///////////
// Structure for CtrlPcs Jema .  
//////////
TYPE PCS_Jema :
STRUCT
// PCS Controller  Measures
	AX_PowerCol					: ARRAY[1..3] OF PowerCol;

	MesData						: PCS ; 
	
END_STRUCT
END_TYPE

(* stored: Version 1.1.0.1, ProductVersion 3.1.4024.6
   DUT PCS_Jema: Id {e14dc06c-e55c-4281-8cf1-e3bfd6fc2aff} *)
